(* PLC project Generated.project, CODESYS CODESYS V3.5 SP19 Patch 1 *)
(* stored: creationDateTime 2026-08-18T12:53:23.540500, modificationDateTime 2026-08-18T12:53:23.540500 *)

(* ═══════════════════════════════════════════════════════════════ ⚙️ ST_WinchHMI — Données d'échange IHM pour un treuil (M1: moteur de retenue / M2: moteur Benne) ─────────────────────────────────────────────────────────────── 🎨 Destiné à l'affichage des bargraphes, LEDs, mesures et réglages. 📄 Structuration en Cmd / State / Cfg / Safety / Bypass ═══════════════════════════════════════════════════════════════ *)
TYPE ST_WinchHMI : STRUCT
  Cmd : ST_WinchCmd;  (* 🎮 Commandes opérateur *)
  State : ST_WinchState;  (* 🚦 États, retours et mesures *)
  Cfg : ST_WinchCfg;  (* Configurations et limites *)
  Safety : ST_SafetyWinch;  (* 🛡️ Sécurité (FB_Safety_Winch) *)
  Bypass : ST_BypassWinch;  (* Bypass maintenance *)
END_STRUCT;
END_TYPE

(* ═══════════════════════════════════════════════════════════════ ST_BypassWinch — Bypass maintenance dédiés à UN treuil (M1 ou M2) ─────────────────────────────────────────────────────────────── 🎨 Regroupe les bypass "dégradé assumé" propres à un axe (codeur, contacteurs) — chaque treuil a son propre matériel, donc son propre struct (imbriqué M1Winch.Bypass / M2Winch.Bypass). 🔒 Doctrine : actionnable UNIQUEMENT en MAINT_N2, RETAIN, jamais masque les autres défauts du même bloc (voir REGISTRE_ACTIONS_Bypass_v1.0 (archive)). ⚠️ Les bypass de capteurs COMMUNS (SlackCable, TopPositionSensor — capteur physique unique partagé M1/M2) sont dans ST_CommunHMI.Bypass, PAS ici. ═══════════════════════════════════════════════════════════════ *)
TYPE ST_BypassWinch : STRUCT
  OperatorComm : BOOL;  (* 📡 1. Communication & Systèmes auxiliaires 📡 Bypass communication esclave CANopen Joystick / heartbeat IHM *)
  EncoderFault : BOOL;  (* 🔌 Bypass diagnostic esclave EtherCAT COD (codeur absolu) *)
  ContactorFeedback : BOOL;  (* 🔌 Bypass feedbacks contacteurs de puissance et frein *)
  PhaseRotation : BOOL;  (* ⚡ Bypass défaut rotation de phases (commun machine) *)
  BrakeThermal : BOOL;  (* 🌡️ Bypass surchauffe thermique frein (commun machine) *)
  MotorThermal : BOOL;  (* : 🌡️ Bypass surchauffe thermique moteur CE treuil (M1_ThermalOk_DI/M2_ThermalOk_DI) *)
  TopLimitSwitch : BOOL;  (* 🚧 2. Limites physiques et Positionnement 🚧 Bypass fin de course physique haute (capteur, bit5) *)
  TopLimitSoftware : BOOL;  (* : Bypass fin de course logiciel haut (position calculée CablePosM >= TopLimitM, symétrique CableLimitSwitch) *)
  CableLimitSwitch : BOOL;  (* 🚧 Bypass limite basse physique (longueur de câble max) *)
  LimitLegal : BOOL;  (* : Bypass limite légale de profondeur (GVL_IHM.Commun.LimitLegalReached) *)
  MecaA : BOOL;  (* ⚙️ 3. Sécurité Mécanique (Méca A-E) 🔄 Bypass Méca A : mouvement non commandé à l'arrêt *)
  MecaB : BOOL;  (* 🛑 Bypass Méca B : absence confirmation arrêt (frein/contacteurs) *)
  MecaC : BOOL;  (* 🏋️ Bypass Méca C : glissement de charge (benne M1) *)
  MecaD : BOOL;  (* 🚧 Bypass Méca D : arrivée butée haute anormale *)
  MecaE : BOOL;  (* 🔄 Bypass Méca E : désynchronisation critique *)
  Safety : BOOL;  (* 🛡️ 4. Hiérarchie & Restauration 🛡️ Bypass groupé : tous les bits qui provoquent un PowerCutOff *)
  Process : BOOL;  (* ⚙️ Bypass groupé : tous les bits qui provoquent un SafeStop *)
  Global : BOOL;  (* 🌐 Bypass Global : ignore toutes les sécurités de cet axe *)
  Initialized : BOOL := FALSE;  (* FIX persistance (voir DOC/AUDITS/ConfigPersistence/) : flag restauration boot dédié (défaut FALSE non ambigu, contrairement à une valeur métier) — PRG_SUPERVISION_CFC.st 🚦 TRUE = bypass restauré depuis GVL_BypassRetain ce boot *)
END_STRUCT;
END_TYPE

(* ═══════════════════════════════════════════════════════════════ 🛡️ ST_SafetyWinch — Diagnostics de sécurité pour un treuil ─────────────────────────────────────────────────────────────── 🎨 Destiné à l'affichage des défauts de sécurité d'un treuil. ═══════════════════════════════════════════════════════════════ *)
TYPE ST_SafetyWinch : STRUCT
  Error : BOOL;  (* 🛡️ Bloc sécurité (Safety) en défaut *)
  ErrorId : WORD;  (* ❌ Code bitfield du défaut de sécurité *)
  SafeStop : BOOL;  (* 🟧 Arrêt rapide activé par la sécurité *)
  DescendPermit : BOOL;  (* 🟢 Descente autorisée (TRUE = OK | FALSE = mou de câble / limite basse) *)
  AscentPermit : BOOL;  (* 🟢 Montée autorisée (TRUE = OK | FALSE = fin de course haut) *)
  SlackCable : BOOL;  (* ⚠️ Mou de câble physiquement détecté *)
  ThermalFault : BOOL;  (* 🔥 Surchauffe thermique moteur *)
  EncoderFault : BOOL;  (* 🔌 Perte de liaison ou incohérence codeur *)
  BypassActive : BOOL;  (* Bypass codeur effectivement accepté, uniquement MAINT_N2 *)
  CableLimitDescent : BOOL;  (* ⚠️ Longueur max de câble atteinte (limite basse physique) *)
  CableLimitAscent : BOOL;  (* ⚠️ Limite haute d'exploitation normale atteinte *)
  MecaADrift_M : REAL;  (* 📐 Dérive mesurée Méca A (m) *)
  MecaCDrift_M : REAL;  (* 📐 Dérive mesurée Méca C (m) *)
  MecaBElapsedTime : TIME;  (* ⏳ Temps écoulé confirmation contacteurs/frein *)
  PowerCutOff : BOOL;  (* 🧨 Coupure puissance amont activée *)
  BlockedBySafety : BOOL;  (* 🚫 Synthèse globale : actionneur bloqué par la sécurité (PowerCutOff OU SafeStop/Error) *)
  PowerCutOffSafety : BOOL;  (* 🧨 Synthèse sécurités critiques entraînant une coupure puissance *)
  SafeStopSafety : BOOL;  (* 🛡️ Synthèse défauts entraînant un SafeStop / Rampe rapide *)
  ErrorOperatorComm : BOOL;  (* 🔍 Décomposition individuelle des défauts de sécurité (bits ErrorId) 🎮 Perte communication opérateur : joystick CAN ou heartbeat IHM (bit0) *)
  ErrorEncoder : BOOL;  (* 🔌 Perte de liaison ou incohérence codeur (bit1) *)
  ErrorPhaseRotation : BOOL;  (* ⚡ Mauvaise rotation de phases électriques (bit4) *)
  ErrorBrakeThermal : BOOL;  (* 🌡️ Surchauffe thermique frein commun M1/M2/M3 (bit10) *)
  ErrorMecaA : BOOL;  (* 🔄 Mouvement non commandé / roue libre (Méca A - bit7) *)
  ErrorMecaB : BOOL;  (* 🛑 Absence confirmation arrêt sans commande (Méca B - bit8) *)
  ErrorMecaC : BOOL;  (* 🏋️ Glissement M1 pendant cycle benne (Méca C - bit9) *)
  ErrorMecaD : BOOL;  (* 🚧 Non-arrêt sur capteur haut (Méca D - bit11) *)
  ErrorMecaE : BOOL;  (* 🔄 Écart de synchronisation critique M1/M2 (Méca E - bit12/13) *)
  ErrorOppositeDir : BOOL;  (* 🧭 Sens réel opposé au sens commandé (bit14) *)
  ErrorNoMovement : BOOL;  (* ⏱️ Absence de mouvement malgré commande (bit15) *)
END_STRUCT;
END_TYPE

(* ═══════════════════════════════════════════════════════════════ ST_WinchCfg — Configurations et paramètres réglables pour un Treuil M1/M2 ─────────────────────────────────────────────────────────────── 🎨 Destiné au paramétrage et calibration depuis l'IHM (RETAIN). 📄 : CfgMaxStepDescente/CfgMaxStepAscent/CfgSlowdownDistance_M/CfgSlowSpeed_Pct déplacés vers GVL_IHM.Commun.Cfg (WinchMaxStepDescente/etc.) — étaient partagés M1/M2 via réconciliation ad-hoc, une seule instance dans Commun élimine le besoin de réconciliation. ═══════════════════════════════════════════════════════════════ *)
TYPE ST_WinchCfg : STRUCT
  CfgTopSensorPos_M : REAL := 8.5;  (* 📐 Position cible du capteur haut (m) *)
  CfgHomingTarget_M : REAL := 0;  (* Cible libre Homing unitaire MAINT_N2 [-99..+99 m] *)
  CfgRampAccelRate : REAL := 50;  (* 📈 Rampe d'accélération (%/s) *)
  CfgRampDecelNormalRate : REAL := 150;  (* 📉 Rampe de décélération normale (%/s) *)
  CfgRampDecelFastRate : REAL := 400;  (* ⚡ Rampe de décélération rapide / SafeStop (%/s) *)
  CfgCableLimitDescent_M : REAL := -20;  (* 📐 Limite basse physique de descente (m, négatif) *)
  CfgCableLimitAscent_M : REAL := 6.75;  (* 📐 Limite haute d'exploitation NORMALE (m) -- (25), aligné sur GVL_PERSISTENT *)
  Initialized : BOOL := FALSE;  (* FIX : flag restauration boot (défaut FALSE non ambigu, contrairement à un champ métier dont le défaut peut valoir n'importe quoi) — PRG_SUPERVISION_CFC.st §2/§3 🚦 TRUE = config restaurée depuis GVL_PERSISTENT ce boot *)
END_STRUCT;
END_TYPE

(* ═══════════════════════════════════════════════════════════════ 🎮 ST_WinchCmd — Commandes IHM pour un Treuil M1/M2 ─────────────────────────────────────────────────────────────── 🎨 Destiné au pilotage manuel et maintenance du treuil depuis l'IHM. ═══════════════════════════════════════════════════════════════ *)
TYPE ST_WinchCmd : STRUCT
  BtnUp : BOOL;  (* ⬆️ Mouvement montee maintenu (mode boutons IHM, MAINT_N1 accessible) *)
  BtnDown : BOOL;  (* ⬇️ Mouvement descente maintenu (mode boutons IHM, MAINT_N1 accessible) *)
  BtnReset : BOOL;  (* 🔑 Demande reset exposée par treuil ; agrégée dans le reset domaine partagé *)
  BtnHome : BOOL;  (* 🎯 Homing nominal si Couplé, unitaire si M1/M2 sélectionné en MAINT_N2 *)
  BtnConfirmCoherence : BOOL;  (* 🔓 Confirmation de cohérence au démarrage *)
  BtnInhibit : BOOL;  (* Bouton IHM inhibition treuil — mise en service, *)
  BtnHomingAtZero : BOOL;  (* Force le homing à 0 m (points codeur centre), *)
END_STRUCT;
END_TYPE

(* ═══════════════════════════════════════════════════════════════ 🚦 ST_WinchState — États, mesures et diagnostics HMI pour un Treuil M1/M2 ─────────────────────────────────────────────────────────────── 🎨 Destiné aux retours d'informations et bargraphes HMI. ═══════════════════════════════════════════════════════════════ *)
TYPE ST_WinchState : STRUCT
  Position_M : REAL;  (* 🚦 États & Mesures (Lecture seule) 📊 Position actuelle du câble (mètres) *)
  MeasuredSpeed_Mps : REAL;  (* 📏 Vitesse linéaire mesurée du câble (m/s), valeur absolue *)
  SpeedDelta_Mps : REAL;  (* 🔍 Variation de vitesse entre deux scans (m/s) *)
  SpeedVariationDetected : BOOL;  (* 🔍 Seuil de variation dépassé sur le scan courant *)
  SpeedVariationConfirmed : BOOL;  (* 🛡️ Variation confirmée pendant la durée paramétrée *)
  SpeedStable : BOOL;  (* 🟢 Vitesse stable pendant la durée paramétrée *)
  SpeedMonitorError : BOOL;  (* Défaut mémorisé du moniteur vitesse *)
  SpeedMonitorErrorId : WORD;  (* ❌ Bitfield du moniteur vitesse *)
  EstimatedLoadPct : REAL;  (* 📊 Estimation empirique, non certifiée *)
  LoadEstimateConfigured : BOOL;  (* 🟢 Table charge validée pour lecture *)
  SpeedGuardLimited : BOOL;  (* 🛡️ Palier limité par vitesse réelle *)
  SpeedRef_Pct : REAL;  (* 📈 Consigne de vitesse finale après rampe (%) *)
  StepNumber : INT;  (* 🔢 Palier de vitesse actif (0..5) *)
  FBState : E_State;  (* 🤖 État de l'automate interne (FB_Winch) *)
  Ready : BOOL;  (* 🟢 Treuil prêt à fonctionner *)
  Busy : BOOL;  (* ⚙️ Mouvement en cours *)
  Done : BOOL;  (* ✅ Action terminée *)
  Error : BOOL;  (* Treuil en défaut *)
  ErrorId : WORD;  (* ❌ Code bitfield du défaut treuil *)
  RelayFwd : BOOL;  (* 🔌 Sorties Physiques / Indicateurs LEDs 🛗 Relais Montée activé *)
  RelayRev : BOOL;  (* 🛗 Relais Descente activé *)
  Contactor1 : BOOL;  (* 🔌 Contacteur vitesse palier 1 *)
  Contactor2 : BOOL;  (* 🔌 Contacteur vitesse palier 2 *)
  Contactor3 : BOOL;  (* 🔌 Contacteur vitesse palier 3 *)
  Contactor4 : BOOL;  (* 🔌 Contacteur vitesse palier 4 *)
  BrakeCmd : BOOL;  (* 🔓 Commande frein (TRUE = desserré / libre) *)
  FinalInterlockState : E_WinchFinalInterlockState;  (* 🛡️ État final _LD lecture seule *)
  FinalInterlockReason : E_WinchFinalInterlockReason;  (* 🛡️ Cause finale mémorisée *)
  FinalInterlockError : BOOL;  (* 🛡️ Défaut final mémorisé *)
  FinalInterlockErrorId : WORD;  (* 🛡️ Bitfield final *)
  FinalRestartInhibit : BOOL;  (* 🔒 Reset + neutre + nouvelle demande obligatoires *)
  BrakeCommandOpenConfirmed : BOOL;  (* 🔌 Contacteur/bobine desserrage confirmé, pas frein mécanique *)
  FinalAuthorizedStep : INT;  (* 🪜 Palier réellement autorisé *)
  FinalBrakeTimeoutElapsed : TIME;  (* ⏱️ Écoulé watchdog 500ms *)
  FinalRestartDelayElapsed : TIME;  (* ⏱️ Écoulé verrou redémarrage 900ms *)
  FinalStepDelayElapsed : TIME;  (* ⏱️ Écoulé entre paliers 1s250 *)
  Encoder : ST_EncoderHMI;  (* 🛡️ Sécurités & Diagnostics 🧲 Données d'échange et diagnostic du codeur — porte aussi les 9 champs Homing* (déplacés 2026-08, voir ST_EncoderHMI) *)
  ContactorsCheck : ST_ContactorCheck;  (* 🔍 Diagnostics de cohérence contacteurs réutilisés 🔌 Coherence contacteurs sens+vitesse *)
  BrakeContactorCheck : ST_ContactorCheck;  (* 🔌 Coherence retour frein *)
  InhibitActive : BOOL;  (* miroir lecture seule — inhibition arbitrée *)
  BottomLimitActiveM : REAL;  (* 🐢 : ralentissement sur bordure — diagnostic zone/limite active 📏 Limite basse active (m) — câble physique OU légale, la plus restrictive *)
  InTopSlowdownZone : BOOL;  (* 🐢 Palier plafonné à 1 : approche limite haute *)
  InBottomSlowdownZone : BOOL;  (* 🐢 Palier plafonné à 1 : approche limite basse (câble ou légale) *)
  CommandedDirection : INT;  (* 🩺 Diagnostic délai ressenti à la remontée 🩺 Sens interne mémorisé FB_Winch (-1/0/+1) *)
  DirectionChangeDelayElapsed : TIME;  (* 🩺 Écoulé de l'interlock changement/reprise de sens *)
  DirectionChangePending : BOOL;  (* 🩺 TRUE tant que CommandedDirection n'a pas rejoint Direction *)
END_STRUCT;
END_TYPE

(* values of E_State: DISABLED: Enable faux, neutralisé; INIT: Démarrage / vérifs; READY: Prêt, attend ordre; BUSY: Action en cours; DONE: Action terminée; STOPPING: Décél rampe avant arrêt (StartStop=FALSE ou SafeStop=TRUE) *)

{attribute 'qualified_only'}
{attribute 'strict'}
TYPE E_State : (DISABLED := 0, INIT := 1, READY := 2, BUSY := 3, DONE := 4, STOPPING := 5);
END_TYPE

(* values of E_WinchFinalInterlockReason: NONE: Aucun blocage actif; BRAKE_COMMAND_NOT_CONFIRMED: Absence confirmation ouverture frein > 500ms; RESTART_INHIBITED: Inhibition redemarrage actif *)

{attribute 'qualified_only'}
{attribute 'strict'}
TYPE E_WinchFinalInterlockReason : (NONE := 0, BRAKE_COMMAND_NOT_CONFIRMED := 1, RESTART_INHIBITED := 2);
END_TYPE

(* values of E_WinchFinalInterlockState: DISABLED: Desactive / Hors service; READY: Pret / Etat nominal; WAIT_BRAKE_COMMAND_CONFIRMATION: Attente confirmation feedback frein; WAIT_STEP_DELAY: Temporisation changement de palier; WAIT_RESTART_DELAY: Temporisation anti-court-cycle redemarrage; FAULT: Etat de defaut *)

{attribute 'qualified_only'}
{attribute 'strict'}
TYPE E_WinchFinalInterlockState : (DISABLED := 0, READY := 1, WAIT_BRAKE_COMMAND_CONFIRMATION := 2, WAIT_STEP_DELAY := 3, WAIT_RESTART_DELAY := 4, FAULT := 5);
END_TYPE

(* ======================================================================= 🔌 ST_ContactorCheck — Double vérification commande/retour contacteur ─────────────────────────────────────────────────────────────── 🎯 Rôle : Structure de diagnostic pour vérification commande vs retour 📊 Diagnostic : Détection des défauts contacteur (StuckClosed / StuckOpen) 📄 Doc métier : DOC/AF/AF_Partie-03_Contrats_Composants_v2.1.md §2 ======================================================================= *)
TYPE ST_ContactorCheck : STRUCT
  Command : BOOL;  (* Ordre envoyé au contacteur (TRUE = fermé/actif) *)
  Feedback : BOOL;  (* Retour d'état câblé (TRUE = effectivement fermé) *)
  StuckClosed : BOOL;  (* Diag : commande OFF mais retour ON depuis trop longtemps → PowerCutOff *)
  StuckOpen : BOOL;  (* Diag : commande ON mais retour OFF depuis trop longtemps *)
END_STRUCT;
END_TYPE

(* ═══════════════════════════════════════════════════════════════ 🧲 ST_EncoderHMI — Données d'échange IHM pour les codeurs absolus ─────────────────────────────────────────────────────────────── 🎨 Destiné à l'affichage des informations et diagnostics des codeurs. ═══════════════════════════════════════════════════════════════ *)
TYPE ST_EncoderHMI : STRUCT
  RawPos : UDINT;  (* 📊 Position brute lue sur le bus *)
  Alarms : UINT;  (* ⚠️ Code d'alarme brut du codeur *)
  Warnings : UINT;  (* 🟧 Code d'avertissement brut du codeur *)
  SlaveOperational : BOOL;  (* 📡 Esclave EtherCAT opérationnel *)
  PresetTriggerCmd : WORD;  (* 🎯 Commande de preset active *)
  PresetValueOut : UDINT;  (* 📐 Valeur de preset envoyée au codeur *)
  Error : BOOL;  (* Codeur en défaut (liaison EtherCAT ou preset) *)
  ErrorId : WORD;  (* ❌ Code défaut codeur *)
  Homed : BOOL;  (* 🎯 Homing — déplacés depuis ST_WinchState racine (2026-08, réorganisation ST_WinchHMI/Homing) 🎯 Prise d'origine (Homing) validée *)
  HomingBusy : BOOL;  (* ⏳ Référencement en cours *)
  HomingDone : BOOL;  (* ✅ Pulse de référencement réussi *)
  HomingError : BOOL;  (* Défaut de référencement *)
  HomingErrorId : WORD;  (* ❌ Bitfield défaut homing *)
  HomingState : E_State;  (* 🤖 État FB_Encoder_Homing *)
  HomingStateAtError : E_State;  (* 🧭 État lors du défaut *)
  HomingSuspect : BOOL;  (* ⚠️ Référence à confirmer *)
  HomingRefRaw : UDINT;  (* 📐 Référence brute appliquée *)
END_STRUCT;
END_TYPE
